PROGRAM Test
VAR
END_VAR

// Feste Geschwindigkeit und Winkel festlegen
GVL_Datatransfer23.gvFahrvektor.reGeschwindigkeit := 100;
GVL_Datatransfer23.gvFahrvektor.reWinkel := 180;

END_PROGRAM

(* stored: Version 1.1.0.1, ProductVersion 3.1.4026.13
   POU Test: Id {45ae4d52-4131-4c96-aad5-0de207b3d4c3}, SpecialFunc None *)
